// SIMATIC S7-200 project (STEP 7-Micro/WIN), CPU 224XP REL 02.01

SYMBOL_TABLE USUARIO1
SENSOR           I0.0     // SENSOR QUE ABRE LA PUERTA
CELULA           I0.1     // CELULA ENCARGADA DE CERRAR LA PUERTA
FCA              I0.2     // FINAL DE CARRERA DE APERTURA
FCC              I0.3     // FINAL DE CARRERA DE CIERRE
APERTURA         Q0.0     // APERTURA DE LA PUERTA
CIERRE           Q0.1     // CIERRE DE L A PUERTA
END_SYMBOL_TABLE

ORGANIZATION_BLOCK PRINCIPAL:OB1
TITLE=APERTURA Y CIERRE DE UN PORTON CON CONTROL DE MOVIMIENTO PARA APERTURA Y CONTROL FOTOELECTRICO PARA EL CIERRE		
BEGIN
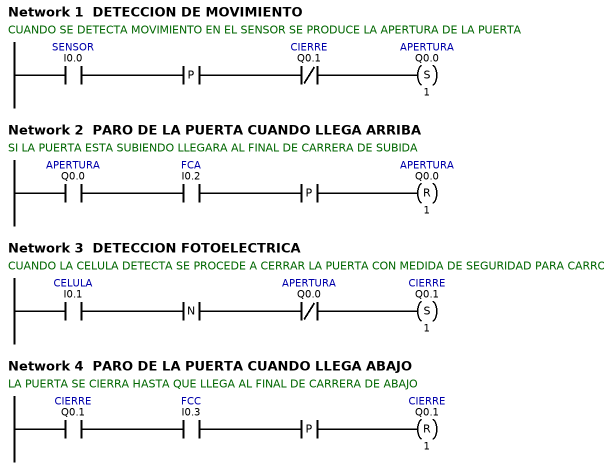
Network 1 // DETECCION DE MOVIMIENTO	
// CUANDO SE DETECTA MOVIMIENTO EN EL SENSOR SE PRODUCE LA APERTURA DE LA PUERTA
LD     SENSOR:I0.0
EU
AN     CIERRE:Q0.1
S      APERTURA:Q0.0, 1
Network 2 // PARO DE LA PUERTA CUANDO LLEGA ARRIBA	
// SI LA PUERTA ESTA SUBIENDO LLEGARA AL FINAL DE CARRERA DE SUBIDA
LD     APERTURA:Q0.0
A      FCA:I0.2
EU
R      APERTURA:Q0.0, 1
Network 3 // DETECCION FOTOELECTRICA
// CUANDO LA CELULA DETECTA SE PROCEDE A CERRAR LA PUERTA CON MEDIDA DE SEGURIDAD PARA CARROS Y PERSONAS UTILIZANDO UN FLANCO NEGATIVO
LD     CELULA:I0.1
ED
AN     APERTURA:Q0.0
S      CIERRE:Q0.1, 1
Network 4 // PARO DE LA PUERTA CUANDO LLEGA ABAJO
// LA PUERTA SE CIERRA HASTA QUE LLEGA AL FINAL DE CARRERA DE ABAJO
LD     CIERRE:Q0.1
A      FCC:I0.3
EU
R      CIERRE:Q0.1, 1
END_ORGANIZATION_BLOCK
